// LS Electric XG5000 project: test
// PLC LSPLC
// module base 0 slot 0: 입출력 모듈:XBC-DR14E (DC 24V 입력 8점, 릴레이 출력 6점)

PROGRAM NewProgram (task: 스캔 프로그램)

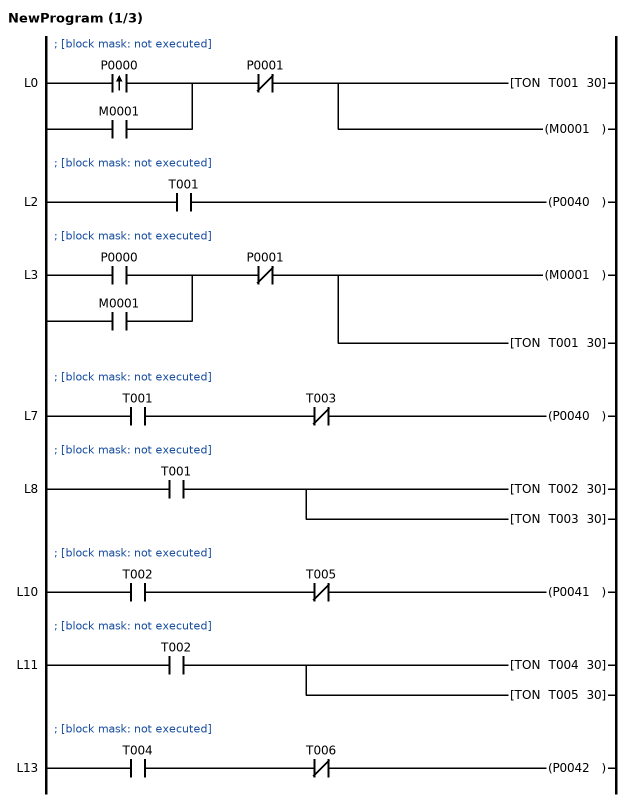
; L0 (block mask: not executed)
LOADP     P0000
OR        M0001
AND NOT   P0001
TON       T001 30
OUT       M0001
; L2 (block mask: not executed)
LOAD      T001
OUT       P0040
; L3 (block mask: not executed)
LOAD      P0000
OR        M0001
AND NOT   P0001
OUT       M0001
TON       T001 30
; L7 (block mask: not executed)
LOAD      T001
AND NOT   T003
OUT       P0040
; L8 (block mask: not executed)
LOAD      T001
TON       T002 30
TON       T003 30
; L10 (block mask: not executed)
LOAD      T002
AND NOT   T005
OUT       P0041
; L11 (block mask: not executed)
LOAD      T002
TON       T004 30
TON       T005 30
; L13 (block mask: not executed)
LOAD      T004
AND NOT   T006
OUT       P0042

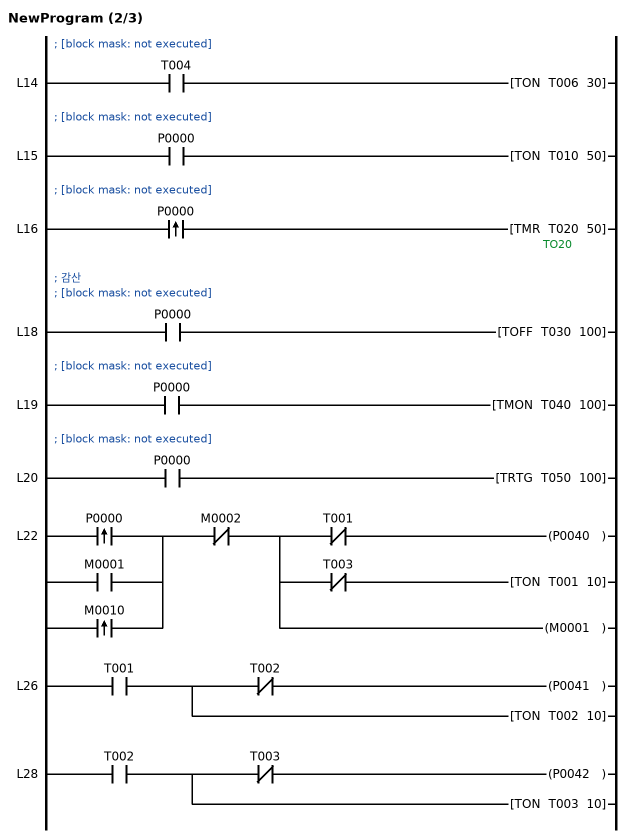
; L14 (block mask: not executed)
LOAD      T004
TON       T006 30
; L15 (block mask: not executed)
LOAD      P0000
TON       T010 50
; L16 (block mask: not executed)
LOADP     P0000
TMR       T020 50	// TO20
// 감산
; L18 (block mask: not executed)
LOAD      P0000
TOFF      T030 100
; L19 (block mask: not executed)
LOAD      P0000
TMON      T040 100
; L20 (block mask: not executed)
LOAD      P0000
TRTG      T050 100
; L22
LOADP     P0000
OR        M0001
ORP       M0010
AND NOT   M0002
MPUSH
AND NOT   T001
OUT       P0040
MLOAD
AND NOT   T003
TON       T001 10
MPOP
OUT       M0001
; L26
LOAD      T001
MPUSH
AND NOT   T002
OUT       P0041
MPOP
TON       T002 10
; L28
LOAD      T002
MPUSH
AND NOT   T003
OUT       P0042
MPOP
TON       T003 10

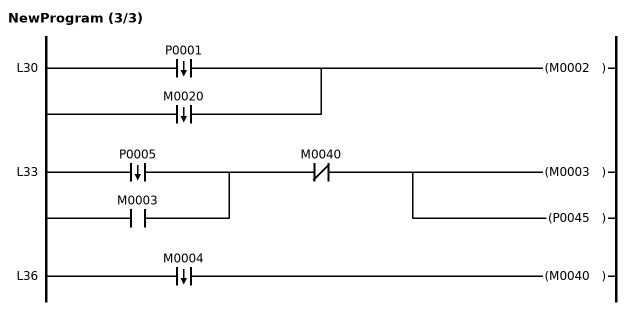
; L30
LOADN     P0001
ORN       M0020
OUT       M0002
; L33
LOADN     P0005
OR        M0003
AND NOT   M0040
OUT       M0003
OUT       P0045
; L36
LOADN     M0004
OUT       M0040